Universal Robots PolyScope program: test1.urp

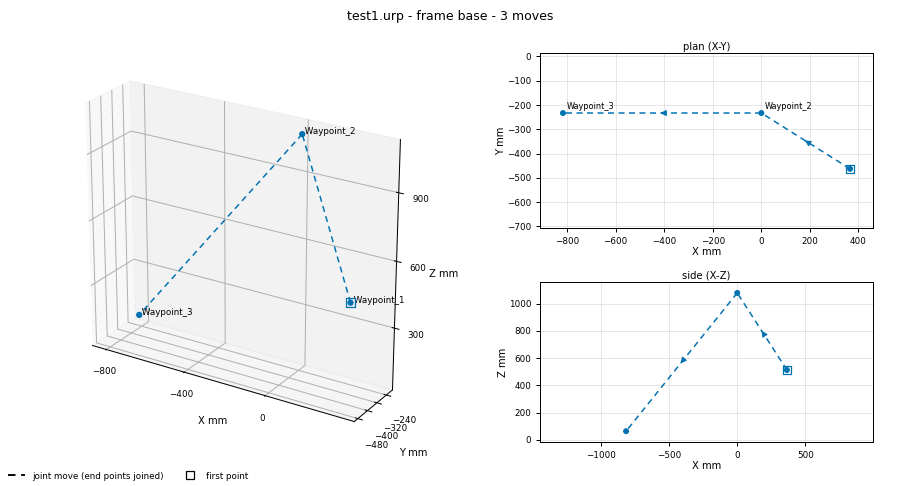
[picture p0: tool path of test1.urp in frame base, 3 of 3 moves have a stored position in this frame; points joined in program order, loops and branches not executed]
Program test1 (installation=default directory=/ursim/programs createdIn=5.14.5 lastSavedIn=5.14.5 robotSerialNumber=20195599999)
Calibrated DH parameters: a=[0, -0.425, -0.3922, 0, 0, 0]; d=[0.1625, 0, 0, 0.1333, 0.0997, 0.0996]; alpha=[1.570796, 0, 0, 1.570796, -1.570796, 0]; deltaTheta=[0, 0, 0, 0, 0, 0]
InitVariablesNode
Robot Program (runOnlyOnce=false)
  MoveJ speed 60 deg/s, acceleration 80 deg/s^2 (useActiveTCP=true positionType=JointAngles) feature=Base
    Waypoint Waypoint_1: TCP in base x=365.378 y=-462.829 z=512.939 mm, rx=-1.1709 ry=2.8335 rz=0.1028 rad; joints [-39.604, -102.063, -72.615, -96.733, 95.543, 5.425] deg
    Waypoint Waypoint_2: TCP in base x=0 y=-232.9 z=1079.4 mm, rx=0 ry=2.2214 rz=-2.2214 rad; joints [0, -90, 0, -90, 0, 0] deg
    Waypoint Waypoint_3: TCP in base x=-817.2 y=-232.9 z=62.8 mm, rx=1.5708 ry=0 rz=0 rad; joints [0, 0, 0, 0, 0, 0] deg
